RoboDK station: Pick and Place.rdk

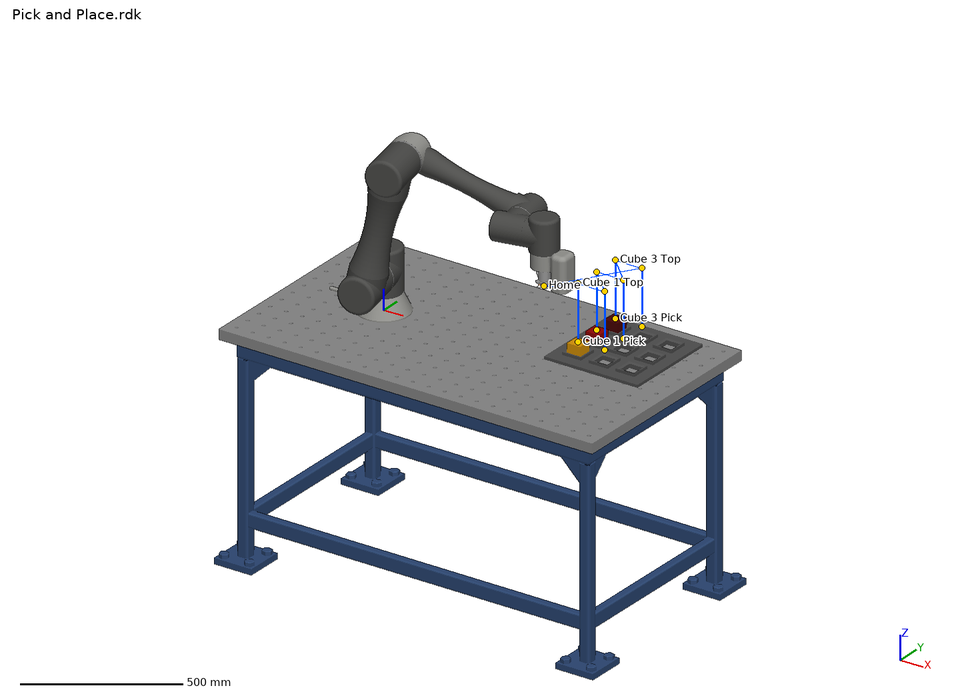
[picture v0: the station drawn from its stored meshes, robots at their saved joint values, targets as dots, program paths as lines]
Station Pick and Place (saved by RoboDK 5.9.2). Poses are relative to the parent item; angles as X-Y-Z fixed-axis rotations.
  - frame TM5-900 Base at (0, 0, 0) mm
    - robot TM5-900: 6 axes, payload 4 kg, reach 900 mm, repeatability 0.1 mm, weight 30 kg
        modified DH rows (alpha deg, a mm, theta deg, d mm): 0, 0, 0, 145.2; 90, 0, 90, 0; 0, 429, 0, 0; 0, 411, -90, 122.3; -90, 0, 0, 106.5; 90, 0, 180, 114.15
        joint limits [-360, -180, -155, -180, -180, -270] to [360, 180, 155, 180, 180, 270]; home [0, 0, 90, -90, 90, 0]; saved at [11.761, 12.588, 96.919, -19.506, 90, 11.761]
      - tool SMC ZXP7A01-ZP25C-X1 Vacuum Gripper, TCP at (0, 0, 62.5) mm, size 44 x 53.4 x 64 mm
    - target Cube 1 Top (Cartesian target) at (675, 75, 250) mm, rotated rx 180 ry 0 rz 90 deg; joints [16.714, 22.857, 83.226, -16.084, 90, 16.714] of TM5-900
    - target Cube 1 Pick (Cartesian target) at (675, 75, 50) mm, rotated rx 180 ry 0 rz 90 deg; joints [16.714, 35.567, 95.041, -40.608, 90, 16.714] of TM5-900
    - target Cube 1 Lift (Cartesian target) at (675, 75, 250) mm, rotated rx 180 ry 0 rz 90 deg; joints [16.714, 22.857, 83.226, -16.084, 90, 16.714] of TM5-900
    - target Cube 1 Push (Cartesian target) at (775, 75, 250) mm, rotated rx 180 ry 0 rz 90 deg; joints [14.565, 36.679, 62.084, -8.762, 90, 14.565] of TM5-900
    - target Cube 1 Place (Cartesian target) at (775, 75, 50) mm, rotated rx 180 ry 0 rz 90 deg; joints [14.565, 46.534, 74.79, -31.324, 90, 14.565] of TM5-900
    - target Cube 1 Release (Cartesian target) at (775, 75, 250) mm, rotated rx 180 ry 0 rz 90 deg; joints [14.565, 36.679, 62.084, -8.762, 90, 14.565] of TM5-900
    - target Cube 2 Top (Cartesian target) at (675, 175, 250) mm, rotated rx 180 ry 0 rz 90 deg; joints [24.636, 25.258, 79.765, -15.023, 90, 24.636] of TM5-900
    - target Cube 2 Pick (Cartesian target) at (675, 175, 50) mm, rotated rx 180 ry 0 rz 90 deg; joints [24.636, 37.463, 91.612, -39.075, 90, 24.636] of TM5-900
    - target Cube 2 Lift (Cartesian target) at (675, 175, 250) mm, rotated rx 180 ry 0 rz 90 deg; joints [24.636, 25.258, 79.765, -15.023, 90, 24.636] of TM5-900
    - target Cube 2 Push (Cartesian target) at (775, 175, 250) mm, rotated rx 180 ry 0 rz 90 deg; joints [21.579, 39.134, 58.038, -7.172, 90, 21.579] of TM5-900
    - target Cube 2 Place (Cartesian target) at (775, 175, 50) mm, rotated rx 180 ry 0 rz 90 deg; joints [21.579, 48.471, 71.123, -29.594, 90, 21.579] of TM5-900
    - target Cube 2 Release (Cartesian target) at (775, 175, 250) mm, rotated rx 180 ry 0 rz 90 deg; joints [21.579, 39.134, 58.038, -7.172, 90, 21.579] of TM5-900
    - target Cube 3 Top (Cartesian target) at (675, 275, 250) mm, rotated rx 180 ry 0 rz 90 deg; joints [31.826, 29.527, 73.384, -12.911, 90, 31.826] of TM5-900
    - target Cube 3 Pick (Cartesian target) at (675, 275, 50) mm, rotated rx 180 ry 0 rz 90 deg; joints [31.826, 40.851, 85.404, -36.254, 90, 31.826] of TM5-900
    - target Cube 3 Lift (Cartesian target) at (675, 275, 250) mm, rotated rx 180 ry 0 rz 90 deg; joints [31.826, 29.527, 73.384, -12.911, 90, 31.826] of TM5-900
    - target Cube 3 Push (Cartesian target) at (775, 275, 250) mm, rotated rx 180 ry 0 rz 90 deg; joints [28.089, 43.754, 50.211, -3.965, 90, 28.089] of TM5-900
    - target Cube 3 Place (Cartesian target) at (775, 275, 50) mm, rotated rx 180 ry 0 rz 90 deg; joints [28.089, 52.062, 64.269, -26.331, 90, 28.089] of TM5-900
    - target Cube 3 Release (Cartesian target) at (775, 275, 250) mm, rotated rx 180 ry 0 rz 90 deg; joints [28.089, 43.754, 50.211, -3.965, 90, 28.089] of TM5-900
    - target Home (Cartesian target) at (600, 0, 250) mm, rotated rx 180 ry 0 rz 90 deg; joints [11.761, 12.588, 96.919, -19.506, 90, 11.761] of TM5-900
  - object Table 1400x800x800mm at (0, 0, 0) mm, size 1420 x 820 x 800 mm, geometry from Table.sld
  - object Pallete  at (600, 0, 0) mm, size 350 x 350 x 20 mm, geometry from Pallete .step
    - object Cube 1 at (50, 50, 0) mm, size 50 x 50 x 50 mm, geometry from Cube.sld
    - object Cube 2 at (50, 150, 0) mm, size 50 x 50 x 50 mm, geometry from Cube.sld
  - program Prog1 (29 instructions, listed below)
  - program Prog2 (1 instructions, listed below)
  - object Cube 3 at (650, 250, 0) mm, size 50 x 50 x 50 mm, geometry from Cube.sld
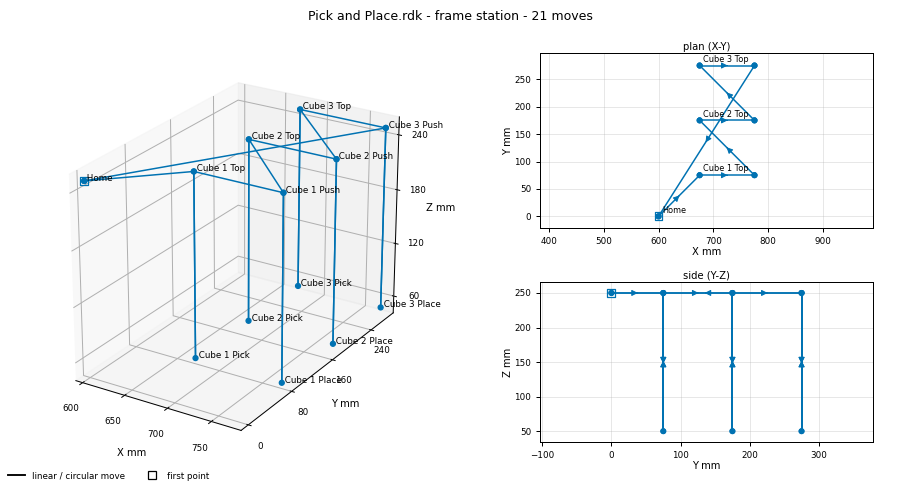
[picture p0: tool path of Pick and Place.rdk in frame station, 21 of 21 moves have a stored position in this frame; points joined in program order, loops and branches not executed]

--- program Prog1 (robot TM5-900) ---
  Set Ref.: TM5-900 Base
  Set Tool: SMC ZXP7A01-ZP25C-X1 Vacuum Gripper at (0, 0, 62.5) mm
  MoveJ (Home)
  MoveL (Home)
  MoveL (Cube 1 Top)
  MoveL (Cube 1 Pick)
  Attach to SMC ZXP7A01-ZP25C-X1 Vacuum Gripper
  MoveL (Cube 1 Lift)
  MoveL (Cube 1 Push)
  MoveL (Cube 1 Place)
  Detach from SMC ZXP7A01-ZP25C-X1 Vacuum Gripper
  MoveL (Cube 1 Release)
  MoveL (Cube 2 Top)
  MoveL (Cube 2 Pick)
  Attach to SMC ZXP7A01-ZP25C-X1 Vacuum Gripper
  MoveL (Cube 2 Lift)
  MoveL (Cube 2 Push)
  MoveL (Cube 2 Place)
  Detach from SMC ZXP7A01-ZP25C-X1 Vacuum Gripper
  MoveL (Cube 2 Release)
  MoveL (Cube 3 Top)
  MoveL (Cube 3 Pick)
  Attach to SMC ZXP7A01-ZP25C-X1 Vacuum Gripper
  MoveL (Cube 3 Lift)
  MoveL (Cube 3 Push)
  MoveL (Cube 3 Place)
  Detach from SMC ZXP7A01-ZP25C-X1 Vacuum Gripper
  MoveL (Cube 3 Release)
  MoveL (Home)

--- program Prog2 (robot TM5-900) ---
  Replace objects
